(* CODESYS project em_log_test.project

Project tree, tasks and I/O mapping:
  Device : EMICON-ARM Cortex-A8-Linux, EMICON, version 3.5.10.0
      settings: IP = '192.168.0.50'
    application Application
      libraries: Standard, * (System); CmpApp, 3.5.11.0 (System); CmpErrors Interfaces, * (System); EmiconLog, 3.5.11.10 (Emicon)
      task MainTask (cyclic, interval t#500ms, priority 1) calls POU, PLC_PRG
      program PLC_PRG [ST]
      program POU [ST]
*)

// Device/Application/POU
PROGRAM POU
VAR
	x: INT;
END_VAR

x := x + 1;

END_PROGRAM

// Device/Application/PLC_PRG
PROGRAM PLC_PRG
VAR
	frame_ti1: ARRAY [1..15] OF BYTE := [16#0,16#0,16#0, 16#0,16#0,16#0,16#0, 16#80, 16#CA,16#1B,16#A6,16#14,16#99,16#08,16#10];
	frame_ti2: ARRAY [1..15] OF BYTE := [16#1,16#0,16#0, 16#0,16#0,16#0,16#0, 16#80, 16#CA,16#1B,16#A6,16#14,16#99,16#08,16#10];
	frame_ts1: ARRAY [1..11] OF BYTE := [16#58,16#0,16#0, 16#80, 16#CA,16#1B,16#A6,16#14,16#99,16#08,16#10];
	frame_ts2: ARRAY [1..11] OF BYTE := [16#59,16#0,16#0, 16#80, 16#CA,16#1B,16#A6,16#14,16#99,16#08,16#10];

	save: BOOL;
	write_log1: BOOL;
	write_log2: BOOL;
	
	cycle : BOOL;
	x : WORD;
	i : BYTE;
	result : UDINT;
	clear: BOOL;
	init: BOOL;
END_VAR

IF NOT init THEN
	EmLog.write_sys_log(3, 11);
	EmLog.write_sys_log(3, 12);
	EmLog.write_sys_log(3, 13);
	init := TRUE;
END_IF

IF write_log1 THEN
	EmLog.write_sys_log(0, 111);
	EmLog.write_sys_log(0, 112);
	EmLog.write_sys_log(0, 113);
	EmLog.write_sys_log(1, 114);
	EmLog.write_sys_log(1, 115);
	EmLog.write_ts_log(3, ADR(frame_ts1[1]));
	EmLog.write_ti_log(45, ADR(frame_ti2[1]));
	write_log1 := FALSE;
END_IF
IF write_log2 THEN
	EmLog.write_sys_log(2, 10);
//	EmLog.write_sys_log(20);
	EmLog.write_ts_log(2, ADR(frame_ts2[1]));
	EmLog.write_ti_log(45, ADR(frame_ti2[1]));
	write_log2 := FALSE;
END_IF

IF save THEN
	EmLog.create_log_files();
	save := FALSE;
END_IF

IF clear THEN
	EmLog.clr_sys_log();
	clear := FALSE;
END_IF


(*
	Проверка записи в цикле.
	При неправильных значениях класса функции записи должны вернуть ошибку.
	write_sys_log - самостоятельно взводит старший бит и значения не проверяет.
	write_tsl_log - Проверяет вхождение класса в список 1, 3, 30, 31
	write_ti_log - Проверяет вхождение класса в список 45, 58

*)

IF cycle THEN
	x := x + 1;
	i := i + 1;
	EmLog.write_sys_log(2, x);
	EmLog.write_ts_log(i, ADR(frame_ts2[1]));
	EmLog.write_ti_log(i, ADR(frame_ti2[1]));	
END_IF

END_PROGRAM
